{attribute 'linkalways'} 
{attribute 'no_explicit_call' := 'This FB is a CLASS and must be accessed using methods or properties'}
{attribute 'enable_dynamic_creation'}
FUNCTION_BLOCK FINAL LE_INT EXTENDS Node
VAR
	in1 : _INT(0);
	in2 : _INT(0);
	out : _BOOL(FALSE);
END_VAR

METHOD PUBLIC Clone : I_Node
VAR
	pNode : POINTER TO LE_INT;
END_VAR
pNode := __NEW(LE_INT);
Clone := pNode^;
END_METHOD

METHOD FB_init : BOOL
VAR_INPUT
	bInitRetains : BOOL; // if TRUE, the retain variables are initialized (warm start / cold start)
	bInCopyCode : BOOL;  // if TRUE, the instance afterwards gets moved into the copy code (online change)
END_VAR
AddInput('in1',THIS^.in1);
AddInput('in2',THIS^.in2);
AddOutput('out', THIS^.out);
END_METHOD

METHOD PROTECTED OnExecute
VAR
END_VAR
out.Value := in1.Value <= in2.Value;
END_METHOD

END_FUNCTION_BLOCK

(* stored: Version 1.1.0.1, ProductVersion 3.1.4024.15
   POU LE_INT: Id {1cbff250-4f5a-45bb-b7a4-bc84520f3eda}, SpecialFunc None
   Folder Constructor: Id {bd16d898-16bd-4ca3-b8f6-c13a799288fa}
   Method Clone: Id {d11bbdec-d7e5-430f-9f7e-9188b8fbcef6}
   Method FB_init: Id {54f640a6-7f26-4c0f-afc8-5bbb4be751fb}
   Method OnExecute: Id {c0ec4fab-f64a-4a4a-939b-9e29976ea836} *)
